INTERFACE I_Enumerator

METHOD PUBLIC Dispose
VAR_INPUT
END_VAR
END_METHOD

METHOD PUBLIC GetValue : BOOL;
VAR_INPUT
	Destination : ANY;
END_VAR
END_METHOD

PROPERTY PUBLIC IsValid : BOOL
GET
END_GET
END_PROPERTY

METHOD PUBLIC MoveNext : BOOL
VAR_INPUT
END_VAR
END_METHOD

END_INTERFACE

(* stored: Version 1.1.0.1, ProductVersion 3.1.4024.12
   Itf I_Enumerator: Id {863b6c67-d871-45ce-9944-b65fd67a74ce}
   Method Dispose: Id {43ce57b6-3744-468b-bb2a-e5cc781a8443}
   Method GetValue: Id {a3aa25e6-2c38-4262-9e4f-b86ff8a4b0bb}
   Property IsValid: Id {16344ffb-9233-434e-beff-c01934548ecd}
   Get Get: Id {f8d2d29d-f068-4b7e-88f4-c9f0ef98bba9}
   Method MoveNext: Id {95a756b9-1053-49ff-8bcf-058296e1437b} *)
